{attribute 'pack_mode' := '0'}


TYPE TrippedInfoData :
    STRUCT
    cntShortCurcuit : DWORD;
    cntOverload     : DWORD;
    cntHWProtect    : DWORD;
    cntOvervolt     : DWORD;
    cntUndervolt    : DWORD;
    remaCoolDown    : WORD;
    maxCurrDragInd  : WORD;
    END_STRUCT
END_TYPE

(* stored: Version 1.1.0.1, ProductVersion 3.1.4022.6
   DUT TrippedInfoData: Id {28aca86c-808c-4464-9665-c431efd90aae} *)
